// TIA Portal V16 export
// export: Created 2020-03-15T18:15:45.2809197Z, ExportSetting WithDefaults, WithReadOnly, DisplayName Totally Integrated Automation Portal, DisplayVersion V16, DisplayName TIA Portal Version Control Interface, DisplayVersion V16, DisplayName TIA Portal Openness, DisplayVersion V16, DisplayName STEP 7 Professional, DisplayVersion V16, DisplayName STEP 7 Safety, DisplayVersion V16, DisplayName WinCC Advanced, DisplayVersion V16
DATA_BLOCK "StepData"   // DB1
{ S7_Optimized_Access := 'TRUE' }
VERSION : 0.1
// stored: AutoNumber true, CodeModifiedDate 2020-03-15T18:10:17.7644754Z, CompileDate 2020-03-15T18:10:18.0143586Z, CreationDate 2020-03-15T11:46:41.4814721Z, DBAccessibleFromOPCUA true, DownloadWithoutReinit false, InterfaceModifiedDate 2020-03-15T18:10:17.7644754Z, IsConsistent true, IsKnowHowProtected false, IsOnlyStoredInLoadMemory false, IsPLCDB false, IsRetainMemResEnabled false, IsWriteProtectedInAS false, MemoryReserve 100, ModifiedDate 2020-03-15T18:10:17.7644754Z, ParameterModified 2020-03-15T18:10:17.7644754Z, StructureModified 2020-03-15T18:10:17.7644754Z
   VAR RETAIN
      Steps : Array[0..99] of "Step";
   END_VAR
   VAR
      Values : "StepValues";
   END_VAR
BEGIN
END_DATA_BLOCK
